// TIA Portal V20 export
FUNCTION "FC_Diagnostic" : Void   // FC2, SCL
{ S7_Optimized_Access := 'TRUE' }
// stored: SetENOAutomatically false
   VAR_INPUT
      bFault1 : Bool;
      bFault2 : Bool;
   END_VAR
   VAR_OUTPUT
      wAlarmWord : Word;
   END_VAR
BEGIN

   #wAlarmWord.%X0 := #bFault1;
   #wAlarmWord.%X1 := #bFault2;
END_FUNCTION
